# B&R Automation Studio project mappView-widget-3dLoader
Automation Studio 


## Logical view

### Program Logical/Program (IEC)

#### Program.st - Cyclic code
```iecst
PROGRAM _INIT
END_PROGRAM

PROGRAM _CYCLIC
	showGrid;
	posX;
	posY;
	posZ;
END_PROGRAM

PROGRAM _EXIT
END_PROGRAM
```

#### Variables.var - Local variables
```iecst
VAR
	posX : REAL;
	posY : REAL;
	posZ : REAL;
	showGrid : BOOL;
END_VAR
```
